Staubli VAL3: getNearestPos.pgx

program getNearestPos(num sio_ID)
  local pointRx currentPosPnt
  local num jDist
  local string jKey
  local num nearestDistance
  local string nearestName
  local string reply
begin
  //**************************************************
  // Identifies the nearest position of those in knownPositions
  // to the current position of the robot.
  //
  // This method is for recovery on, e.g. interlock breaking,
  // to allow a reset to stable working.
  //**************************************************
  currentPosPnt = jointToPoint(flange, world, herej())

  // nearestJ was also going to be returned, but the plan changed.
  // It is retained in case it is sometime useful.
  //nearestJ = origin
  nearestName = "unknown"
  nearestDistance = 1000000

  // Loop through all the positions in knownPositions, checking which has the smallest distance
  jKey = first(knownPositions)
  while jKey != ""
    jDist = distance(currentPosPnt, jointToPoint(flange,world, knownPositions[jKey]))
    if jDist < nearestDistance
      nearestName = jKey
      //nearestJ = knownPositions[jKey]
      nearestDistance = jDist
    endIf
    jKey = next(knownPositions[jKey])
  endWhile

  // Report the closest distance in the form getCurrentPosition:#DIST0.123#POS_gatePosition;
  reply = "getCurrentPosition:#DIST" + toString(".2", nearestDistance) + "#POS_" + nearestName
  taskCreate "sendStatus",10,sendStatus(reply, sio_ID)
end
